/// calibration that is determined by calibration sequences of the unit (static offsets, shifts)
TYPE MoverDataCalibration :
STRUCT
END_STRUCT
END_TYPE

(* stored: Version 1.1.0.1
   DUT MoverDataCalibration: Id {b1e1d72c-6998-49ab-8d08-8043ab9d55f9} *)
